% RSLogix 500 project street light  project.RSS, saved by version 8.30.00.16 %
PROJECT "UNTITLED"    % processor: Bul.1763 MicroLogix 1100 Series A %

PROGRAM FILES
  LAD 2   13 rungs

DATA FILES
  O0 OUTPUT  4 elements
  I1 INPUT  6 elements
  S2 STATUS  66 elements
  B3 BINARY  16 elements
  T4 TIMER  6 elements
  C5 COUNTER  3 elements
  R6 CONTROL  1 elements
  N7 INTEGER  15 elements
  F8 FLOAT  1 elements

LADDER 2
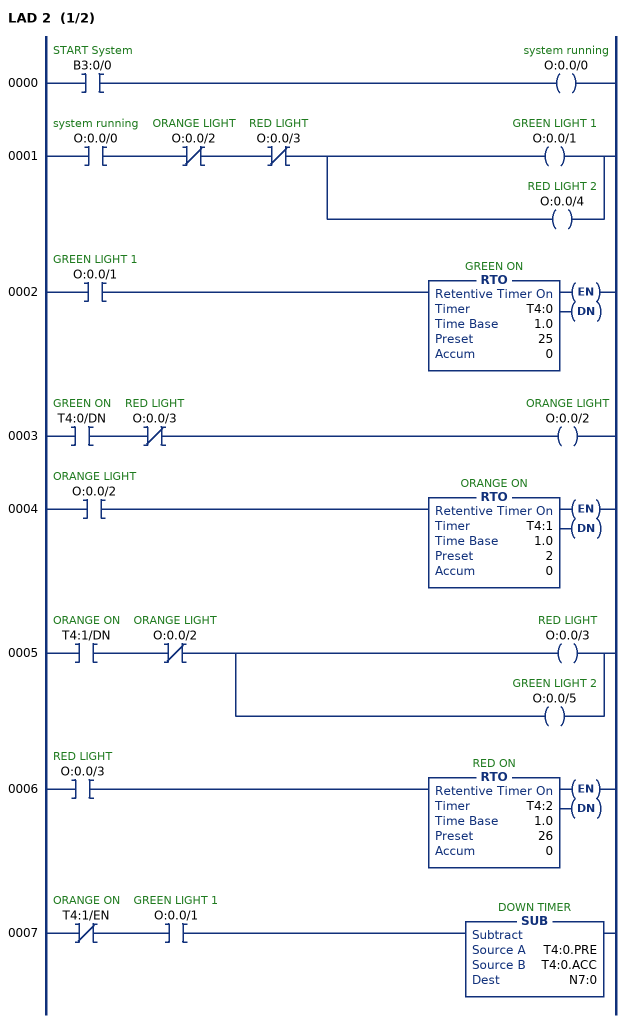
% Rung: 0 %
SOR XIC B3:0/0 OTE O:0.0/0 EOR
%   B3:0/0  "START System" %
%   O:0.0/0  "system running" %
% Rung: 1 %
SOR XIC O:0.0/0 XIO O:0.0/2 XIO O:0.0/3 BST OTE O:0.0/1 NXB OTE O:0.0/4 BND EOR
%   O:0.0/0  "system running" %
%   O:0.0/2  "ORANGE LIGHT" %
%   O:0.0/3  "RED LIGHT" %
%   O:0.0/1  "GREEN LIGHT 1" %
%   O:0.0/4  "RED LIGHT 2" %
% Rung: 2 %
SOR XIC O:0.0/1 RTO T4:0 1.0 25 0 EOR
%   O:0.0/1  "GREEN LIGHT 1" %
%   T4:0  "GREEN ON" %
% Rung: 3 %
SOR XIC T4:0/DN XIO O:0.0/3 OTE O:0.0/2 EOR
%   T4:0  "GREEN ON" %
%   O:0.0/3  "RED LIGHT" %
%   O:0.0/2  "ORANGE LIGHT" %
% Rung: 4 %
SOR XIC O:0.0/2 RTO T4:1 1.0 2 0 EOR
%   O:0.0/2  "ORANGE LIGHT" %
%   T4:1  "ORANGE ON" %
% Rung: 5 %
SOR XIC T4:1/DN XIO O:0.0/2 BST OTE O:0.0/3 NXB OTE O:0.0/5 BND EOR
%   T4:1  "ORANGE ON" %
%   O:0.0/2  "ORANGE LIGHT" %
%   O:0.0/3  "RED LIGHT" %
%   O:0.0/5  "GREEN LIGHT 2" %
% Rung: 6 %
SOR XIC O:0.0/3 RTO T4:2 1.0 26 0 EOR
%   O:0.0/3  "RED LIGHT" %
%   T4:2  "RED ON" %
% Rung: 7 %
SOR XIO T4:1/EN XIC O:0.0/1 SUB T4:0.PRE T4:0.ACC N7:0 EOR
%   T4:1  "ORANGE ON" %
%   O:0.0/1  "GREEN LIGHT 1" %
%   T4:0  "GREEN ON" %
%   N7:0  "DOWN TIMER" %

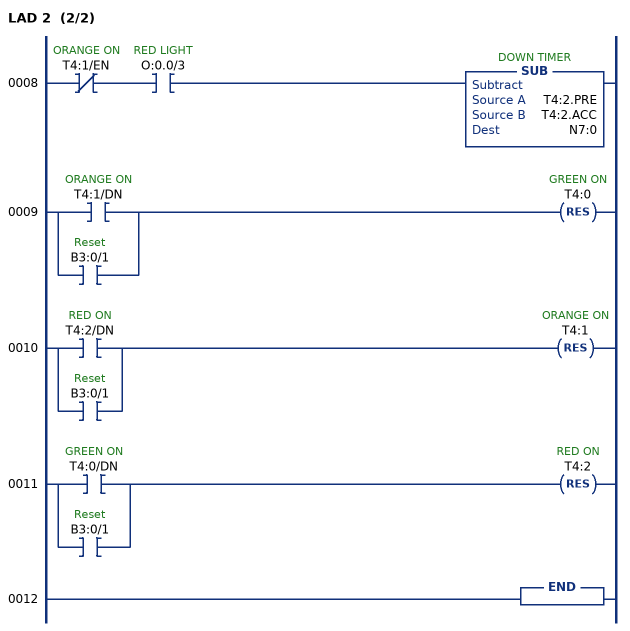
% Rung: 8 %
SOR XIO T4:1/EN XIC O:0.0/3 SUB T4:2.PRE T4:2.ACC N7:0 EOR
%   T4:1  "ORANGE ON" %
%   O:0.0/3  "RED LIGHT" %
%   T4:2  "RED ON" %
%   N7:0  "DOWN TIMER" %
% Rung: 9 %
SOR BST XIC T4:1/DN NXB XIC B3:0/1 BND RES T4:0 EOR
%   T4:1  "ORANGE ON" %
%   B3:0/1  "Reset" %
%   T4:0  "GREEN ON" %
% Rung: 10 %
SOR BST XIC T4:2/DN NXB XIC B3:0/1 BND RES T4:1 EOR
%   T4:2  "RED ON" %
%   B3:0/1  "Reset" %
%   T4:1  "ORANGE ON" %
% Rung: 11 %
SOR BST XIC T4:0/DN NXB XIC B3:0/1 BND RES T4:2 EOR
%   T4:0  "GREEN ON" %
%   B3:0/1  "Reset" %
%   T4:2  "RED ON" %
% Rung: 12 %
SOR END EOR

OTHER DOCUMENTED ADDRESSES
  I:0.0/0  "START"
  N7:1  "downtime red"

DATA TABLE (non-zero values as saved)
DATA T4
% .PRE .ACC %
% T4:0 % 25 0
% T4:1 % 2 0
% T4:2 % 26 0
% T4:3 % 20 0
% T4:5 % 10 0
DATA C5
% .PRE .ACC %
% C5:0 % 20 19
% C5:1 % 5 2
% C5:2 % 20 10
DATA N7
% N7:0 % 0 10 0 0 0 0 0 0 0 0
